// SIMATIC S7-200 project (STEP 7-Micro/WIN), CPU 224 REL 01.11

ORGANIZATION_BLOCK 主:OB1
TITLE=这个项目是基于CPU224的工业脉冲除尘控制系统。已经被实际应用于现实水泥厂布袋除尘器，提供给大家当福利了。
// 系统支持手动和自动两种喷吹模式，分别由I0.0和I0.1控制，手动和自动模式不能同时启用。
// 系统控制的物理设备包括手动喷吹启动按钮、自动喷吹启动按钮、喷吹模式选择开关、喷吹参数选择开关和多个脉冲阀。
// 操作员可以通过手动喷吹启动按钮触发一次手动喷吹，或者按下自动喷吹启动按钮进入自动喷吹模式。不过，手动喷吹启动按钮和自动喷吹启动按钮设计上需避免同时按下，以确保模式切换清晰且操作安全。当两个按钮都未按下时，所有脉冲阀保持关闭，系统停止喷吹，防止意外运行。
// 操作员还可以通过喷吹模式选择开关1、喷吹模式选择开关2和喷吹模式选择开关3的组合，将喷吹时间参数设置为2到9之间的特定值；通过喷吹参数选择开关1、喷吹参数选择开关2和喷吹参数选择开关3的组合，将喷吹间隔参数设置为61到201之间的特定值。喷吹时间参数和喷吹间隔参数分别控制每个脉冲阀的开启时间和阀门之间的等待时间。例如，在手动模式下，按下手动喷吹启动按钮后，系统从脉冲阀1到脉冲阀28依次喷吹，每个阀门按喷吹时间参数开启，间隔由喷吹间隔参数决定。系统通过喷吹状态保持继电器1至喷吹状态保持继电器53管理喷吹过程中的状态转换，确保顺序执行。
// 在自动模式下，系统启动后从脉冲阀1到脉冲阀28完成一次喷吹，周期结束后所有喷吹状态保持继电器和脉冲阀自动复位。而在任一模式下，喷吹完成后，所有喷吹状态保持继电器和脉冲阀都会复位，以保持系统状态的正确性。在手动模式下，喷吹周期完成后，所有喷吹状态保持继电器和脉冲阀复位，等待手动喷吹启动按钮的下一次触发。
// 
//  
BEGIN
Network 1 // 网络题目 (单行)
//  
// 网络注释
//  
// 
LD     SM0.1
R      M0.0, 60
R      T37, 26
R      T101, 30
R      Q0.0, 32
Network 2
LD     I0.0
AN     I0.1
CALL   SBR_0:SBR1
Network 3
LD     I0.1
AN     I0.0
CALL   SBR_1:SBR0
Network 4
LDN    I0.0
AN     I0.1
LPS
R      M0.0, 60
R      Q0.0, 32
R      T37, 26
R      T101, 30
AN     I0.2
AN     I0.3
A      I0.4
MOVW   +2, VW50
LRD
AN     I0.5
AN     I0.6
A      I0.7
MOVW   +61, VW52
LRD
AN     I0.2
A      I0.3
AN     I0.4
MOVW   +3, VW50
LRD
AN     I0.5
A      I0.6
AN     I0.7
MOVW   +81, VW52
LRD
AN     I0.2
A      I0.3
A      I0.4
MOVW   +4, VW50
LRD
AN     I0.5
A      I0.6
A      I0.7
MOVW   +101, VW52
LRD
A      I0.2
AN     I0.3
AN     I0.4
MOVW   +5, VW50
LRD
A      I0.5
AN     I0.6
AN     I0.7
MOVW   +121, VW52
LRD
A      I0.2
AN     I0.3
A      I0.4
MOVW   +6, VW50
LRD
A      I0.5
AN     I0.6
A      I0.7
MOVW   +141, VW52
LRD
A      I0.2
A      I0.3
AN     I0.4
MOVW   +7, VW50
LRD
A      I0.5
A      I0.6
AN     I0.7
MOVW   +161, VW52
LRD
A      I0.2
A      I0.3
A      I0.4
MOVW   +8, VW50
LPP
A      I0.5
A      I0.6
A      I0.7
MOVW   +181, VW52
Network 5
LDN    I0.0
AN     I0.1
LPS
AN     I0.2
AN     I0.3
AN     I0.4
MOVW   +9, VW50
LPP
AN     I0.5
AN     I0.6
AN     I0.7
MOVW   +201, VW52
END_ORGANIZATION_BLOCK

SUBROUTINE_BLOCK SBR_1:SBR0
TITLE= 
// 子程序注释
// 按 F1 获得帮助及举例程序
//  
BEGIN
Network 1 // 网络题目 (单行)
//  
// 网络注释
//  
// 
LD     I0.1
AN     M0.0
R      Q0.0, 28
S      Q0.0, 1
S      M0.0, 1
Network 2
LD     M0.0
A      Q0.0
TON    T37, VW50
Network 3
LDN    M0.1
A      T37
R      Q0.0, 1
R      T37, 1
S      M0.1, 1
Network 4
LD     M0.1
AN     Q0.0
TON    T101, VW52
Network 5
LD     T101
AN     M0.2
R      M0.1, 1
R      T101, 1
S      Q0.1, 1
S      M0.2, 1
Network 6
LD     M0.2
A      Q0.1
TON    T38, VW50
Network 7
LDN    M0.3
A      T38
R      Q0.1, 1
R      T38, 1
S      M0.3, 1
Network 8
LD     M0.3
AN     Q0.1
TON    T102, VW52
Network 9
LD     T102
AN     M0.4
R      M0.3, 1
R      T102, 1
S      Q0.2, 1
S      M0.4, 1
Network 10
LD     M0.4
A      Q0.2
TON    T39, VW50
Network 11
LDN    M0.5
A      T39
R      Q0.2, 1
R      T39, 1
S      M0.5, 1
Network 12
LD     M0.5
AN     Q0.2
TON    T103, VW52
Network 13
LD     T103
AN     M0.6
R      M0.5, 1
R      T103, 1
S      Q0.3, 1
S      M0.6, 1
Network 14
LD     M0.6
A      Q0.3
TON    T40, VW50
Network 15
LDN    M0.7
A      T40
R      Q0.3, 1
R      T40, 1
S      M0.7, 1
Network 16
LD     M0.7
AN     Q0.3
TON    T104, VW52
Network 17
LD     T104
AN     M1.0
R      M0.7, 1
R      T104, 1
S      Q0.4, 1
S      M1.0, 1
Network 18
LD     M1.0
A      Q0.4
TON    T41, VW50
Network 19
LDN    M1.1
A      T41
R      Q0.4, 1
R      T41, 1
S      M1.1, 1
Network 20
LD     M1.1
AN     Q0.4
TON    T105, VW52
Network 21
LD     T105
AN     M1.2
R      M1.1, 1
R      T105, 1
S      Q0.5, 1
S      M1.2, 1
Network 22
LD     M1.2
A      Q0.5
TON    T42, VW50
Network 23
LDN    M1.3
A      T42
R      Q0.5, 1
R      T42, 1
S      M1.3, 1
Network 24
LD     M1.3
AN     Q0.5
TON    T106, VW52
Network 25
LD     T106
AN     M1.6
R      M1.3, 1
R      T106, 1
S      Q0.6, 1
S      M1.6, 1
Network 26
LD     M1.6
A      Q0.6
TON    T43, VW50
Network 27
LDN    M1.7
A      T43
R      Q0.6, 1
R      T43, 1
S      M1.7, 1
Network 28
LD     M1.7
AN     Q0.6
TON    T107, VW52
Network 29
LD     T107
AN     M2.0
R      M1.7, 1
R      T107, 1
S      Q0.7, 1
S      M2.0, 1
Network 30
LD     M2.0
A      Q0.7
TON    T44, VW50
Network 31
LDN    M2.1
A      T44
R      Q0.7, 1
R      T44, 1
S      M2.1, 1
Network 32
LD     M2.1
AN     Q0.7
TON    T108, VW52
Network 33
LD     T108
AN     M2.2
R      M2.1, 1
R      T108, 1
S      Q1.0, 1
S      M2.2, 1
Network 34
LD     M2.2
A      Q1.0
TON    T45, VW50
Network 35
LDN    M2.3
A      T45
R      Q1.0, 1
R      T45, 1
S      M2.3, 1
Network 36
LD     M2.3
AN     Q1.0
TON    T109, VW52
Network 37
LD     T109
AN     M2.4
R      M2.3, 1
R      T109, 1
S      Q1.1, 1
S      M2.4, 1
Network 38
LD     M2.4
A      Q1.1
TON    T46, VW50
Network 39
LDN    M2.5
A      T46
R      Q1.1, 1
R      T46, 1
S      M2.5, 1
Network 40
LD     M2.5
AN     Q1.1
TON    T110, VW52
Network 41
LD     T110
AN     M2.6
R      M2.5, 1
R      T110, 1
S      Q2.0, 1
S      M2.6, 1
Network 42
LD     M2.6
A      Q2.0
TON    T47, VW50
Network 43
LDN    M2.7
A      T47
R      Q2.0, 1
R      T47, 1
S      M2.7, 1
Network 44
LD     M2.7
AN     Q2.0
TON    T111, VW52
Network 45
LD     T111
AN     M3.0
R      M2.7, 1
R      T111, 1
S      Q2.1, 1
S      M3.0, 1
Network 46
LD     M3.0
A      Q2.1
TON    T48, VW50
Network 47
LDN    M3.1
A      T48
R      Q2.1, 1
R      T48, 1
S      M3.1, 1
Network 48
LD     M3.1
AN     Q2.1
TON    T112, VW52
Network 49
LD     T112
AN     M3.2
R      M3.1, 1
R      T112, 1
S      Q2.2, 1
S      M3.2, 1
Network 50
LD     M3.2
A      Q2.2
TON    T49, VW50
Network 51
LDN    M3.3
A      T49
R      Q2.2, 1
R      T49, 1
S      M3.3, 1
Network 52
LD     M3.3
AN     Q2.2
TON    T113, VW52
Network 53
LD     T113
AN     M3.4
R      M3.3, 1
R      T113, 1
S      Q2.3, 1
S      M3.4, 1
Network 54
LD     M3.4
A      Q2.3
TON    T50, VW50
Network 55
LDN    M3.5
A      T50
R      Q2.3, 1
R      T50, 1
S      M3.5, 1
Network 56
LD     M3.5
AN     Q2.3
TON    T114, VW52
Network 57
LD     T114
AN     M3.6
R      M3.5, 1
R      T114, 1
S      Q2.4, 1
S      M3.6, 1
Network 58
LD     M3.6
A      Q2.4
TON    T51, VW50
Network 59
LDN    M3.7
A      T51
R      Q2.4, 1
R      T51, 1
S      M3.7, 1
Network 60
LD     M3.7
AN     Q2.4
TON    T115, VW52
Network 61
LD     T115
AN     M4.0
R      M3.7, 1
R      T115, 1
S      Q2.5, 1
S      M4.0, 1
Network 62
LD     M4.0
A      Q2.5
TON    T52, VW50
Network 63
LDN    M4.1
A      T52
R      Q2.5, 1
R      T52, 1
S      M4.1, 1
Network 64
LD     M4.1
AN     Q2.5
TON    T116, VW52
Network 65
LD     T116
AN     M4.2
R      M4.1, 1
R      T116, 1
S      Q2.6, 1
S      M4.2, 1
Network 66
LD     M4.2
A      Q2.6
TON    T53, VW50
Network 67
LDN    M4.3
A      T53
R      Q2.6, 1
R      T53, 1
S      M4.3, 1
Network 68
LD     M4.3
AN     Q2.6
TON    T117, VW52
Network 69
LD     T117
AN     M4.4
R      M4.3, 1
R      T117, 1
S      Q2.7, 1
S      M4.4, 1
Network 70
LD     M4.4
A      Q2.7
TON    T54, VW50
Network 71
LDN    M4.5
A      T54
R      Q2.7, 1
R      T54, 1
S      M4.5, 1
Network 72
LD     M4.5
AN     Q2.7
TON    T118, VW52
Network 73
LD     T118
AN     M4.6
R      M4.5, 1
R      T118, 1
S      Q3.0, 1
S      M4.6, 1
Network 74
LD     M4.6
A      Q3.0
TON    T55, VW50
Network 75
LDN    M4.7
A      T55
R      Q3.0, 1
R      T55, 1
S      M4.7, 1
Network 76
LD     M4.7
AN     Q3.0
TON    T119, VW52
Network 77
LD     T119
AN     M5.0
R      M4.7, 1
R      T119, 1
S      Q3.1, 1
S      M5.0, 1
Network 78
LD     M5.0
A      Q3.1
TON    T56, VW50
Network 79
LDN    M5.1
A      T56
R      Q3.1, 1
R      T56, 1
S      M5.1, 1
Network 80
LD     M5.1
AN     Q3.1
TON    T120, VW52
Network 81
LD     T120
AN     M5.2
R      M5.1, 1
R      T120, 1
S      Q3.2, 1
S      M5.2, 1
Network 82
LD     M5.2
A      Q3.2
TON    T57, VW50
Network 83
LDN    M5.3
A      T57
R      Q3.2, 1
R      T57, 1
S      M5.3, 1
Network 84
LD     M5.3
AN     Q3.2
TON    T121, VW52
Network 85
LD     T121
AN     M5.4
R      M5.3, 1
R      T121, 1
S      Q3.3, 1
S      M5.4, 1
Network 86
LD     M5.4
A      Q3.3
TON    T58, VW50
Network 87
LDN    M5.5
A      T58
R      Q3.3, 1
R      T58, 1
S      M5.5, 1
Network 88
LD     M5.5
AN     Q3.3
TON    T122, VW52
Network 89
LD     T122
AN     M5.6
R      M5.5, 1
R      T122, 1
S      M5.6, 1
S      Q3.4, 1
Network 90
LD     M5.6
A      Q3.4
TON    T59, VW50
Network 91
LDN    M5.7
A      T59
R      Q3.4, 1
R      T59, 1
S      M5.7, 1
Network 92
LD     M5.7
AN     Q3.4
TON    T123, VW52
Network 93
LD     T123
AN     M6.0
R      M5.7, 1
R      T123, 1
S      M6.0, 1
S      Q3.5, 1
Network 94
LD     M6.0
A      Q3.5
TON    T60, VW50
Network 95
LDN    M6.1
A      T60
R      Q3.5, 1
R      T60, 1
S      M6.1, 1
Network 96
LD     M6.1
AN     Q3.5
TON    T124, VW52
Network 97
LD     T124
AN     M6.2
R      M6.1, 1
R      T124, 1
S      M6.2, 1
S      Q3.6, 1
Network 98
LD     M6.2
A      Q3.6
TON    T61, VW50
Network 99
LDN    M6.3
A      T61
R      Q3.6, 1
R      T61, 1
S      M6.3, 1
Network 100
LD     M6.3
AN     Q3.6
TON    T125, VW52
Network 101
LD     T125
AN     M6.4
R      M6.3, 1
R      T125, 1
S      M6.4, 1
Network 102
LD     M6.4
R      M0.0, 53
R      Q0.0, 32
R      M6.4, 1
END_SUBROUTINE_BLOCK

SUBROUTINE_BLOCK SBR_0:SBR1
TITLE=
BEGIN
Network 1
LD     I0.0
AN     M0.0
R      Q0.0, 28
S      Q0.0, 1
S      M0.0, 1
Network 2
LD     M0.0
A      Q0.0
TON    T37, VW50
Network 3
LDN    M0.1
A      T37
R      Q0.0, 1
R      T37, 1
S      M0.1, 1
Network 4
LD     M0.1
AN     Q0.0
TON    T101, VW52
Network 5
LD     T101
AN     M0.2
R      M0.1, 1
R      T101, 1
S      Q0.1, 1
S      M0.2, 1
Network 6
LD     M0.2
A      Q0.1
TON    T38, VW50
Network 7
LDN    M0.3
A      T38
R      Q0.1, 1
R      T38, 1
S      M0.3, 1
Network 8
LD     M0.3
AN     Q0.1
TON    T102, VW52
Network 9
LD     T102
AN     M0.4
R      M0.3, 1
R      T102, 1
S      Q0.2, 1
S      M0.4, 1
Network 10
LD     M0.4
A      Q0.2
TON    T39, VW50
Network 11
LDN    M0.5
A      T39
R      Q0.2, 1
R      T39, 1
S      M0.5, 1
Network 12
LD     M0.5
AN     Q0.2
TON    T103, VW52
Network 13
LD     T103
AN     M0.6
R      M0.5, 1
R      T103, 1
S      Q0.3, 1
S      M0.6, 1
Network 14
LD     M0.6
A      Q0.3
TON    T40, VW50
Network 15
LDN    M0.7
A      T40
R      Q0.3, 1
R      T40, 1
S      M0.7, 1
Network 16
LD     M0.7
AN     Q0.3
TON    T104, VW52
Network 17
LD     T104
AN     M1.0
R      M0.7, 1
R      T104, 1
S      Q0.4, 1
S      M1.0, 1
Network 18
LD     M1.0
A      Q0.4
TON    T41, VW50
Network 19
LDN    M1.1
A      T41
R      Q0.4, 1
R      T41, 1
S      M1.1, 1
Network 20
LD     M1.1
AN     Q0.4
TON    T105, VW52
Network 21
LD     T105
AN     M1.2
R      M1.1, 1
R      T105, 1
S      Q0.5, 1
S      M1.2, 1
Network 22
LD     M1.2
A      Q0.5
TON    T42, VW50
Network 23
LDN    M1.3
A      T42
R      Q0.5, 1
R      T42, 1
S      M1.3, 1
Network 24
LD     M1.3
AN     Q0.5
TON    T106, VW52
Network 25
LD     T106
AN     M1.6
R      M1.3, 1
R      T106, 1
S      Q0.6, 1
S      M1.6, 1
Network 26
LD     M1.6
A      Q0.6
TON    T43, VW50
Network 27
LDN    M1.7
A      T43
R      Q0.6, 1
R      T43, 1
S      M1.7, 1
Network 28
LD     M1.7
AN     Q0.6
TON    T107, VW52
Network 29
LD     T107
AN     M2.0
R      M1.7, 1
R      T107, 1
S      Q0.7, 1
S      M2.0, 1
Network 30
LD     M2.0
A      Q0.7
TON    T44, VW50
Network 31
LDN    M2.1
A      T44
R      Q0.7, 1
R      T44, 1
S      M2.1, 1
Network 32
LD     M2.1
AN     Q0.7
TON    T108, VW52
Network 33
LD     T108
AN     M2.2
R      M2.1, 1
R      T108, 1
S      Q1.0, 1
S      M2.2, 1
Network 34
LD     M2.2
A      Q1.0
TON    T45, VW50
Network 35
LDN    M2.3
A      T45
R      Q1.0, 1
R      T45, 1
S      M2.3, 1
Network 36
LD     M2.3
AN     Q1.0
TON    T109, VW52
Network 37
LD     T109
AN     M2.4
R      M2.3, 1
R      T109, 1
S      Q1.1, 1
S      M2.4, 1
Network 38
LD     M2.4
A      Q1.1
TON    T46, VW50
Network 39
LDN    M2.5
A      T46
R      Q1.1, 1
R      T46, 1
S      M2.5, 1
Network 40
LD     M2.5
AN     Q1.1
TON    T110, VW52
Network 41
LD     T110
AN     M2.6
R      M2.5, 1
R      T110, 1
S      Q2.0, 1
S      M2.6, 1
Network 42
LD     M2.6
A      Q2.0
TON    T47, VW50
Network 43
LDN    M2.7
A      T47
R      Q2.0, 1
R      T47, 1
S      M2.7, 1
Network 44
LD     M2.7
AN     Q2.0
TON    T111, VW52
Network 45
LD     T111
AN     M3.0
R      M2.7, 1
R      T111, 1
S      Q2.1, 1
S      M3.0, 1
Network 46
LD     M3.0
A      Q2.1
TON    T48, VW50
Network 47
LDN    M3.1
A      T48
R      Q2.1, 1
R      T48, 1
S      M3.1, 1
Network 48
LD     M3.1
AN     Q2.1
TON    T112, VW52
Network 49
LD     T112
AN     M3.2
R      M3.1, 1
R      T112, 1
S      Q2.2, 1
S      M3.2, 1
Network 50
LD     M3.2
A      Q2.2
TON    T49, VW50
Network 51
LDN    M3.3
A      T49
R      Q2.2, 1
R      T49, 1
S      M3.3, 1
Network 52
LD     M3.3
AN     Q2.2
TON    T113, VW52
Network 53
LD     T113
AN     M3.4
R      M3.3, 1
R      T113, 1
S      Q2.3, 1
S      M3.4, 1
Network 54
LD     M3.4
A      Q2.3
TON    T50, VW50
Network 55
LDN    M3.5
A      T50
R      Q2.3, 1
R      T50, 1
S      M3.5, 1
Network 56
LD     M3.5
AN     Q2.3
TON    T114, VW52
Network 57
LD     T114
AN     M3.6
R      M3.5, 1
R      T114, 1
S      Q2.4, 1
S      M3.6, 1
Network 58
LD     M3.6
A      Q2.4
TON    T51, VW50
Network 59
LDN    M3.7
A      T51
R      Q2.4, 1
R      T51, 1
S      M3.7, 1
Network 60
LD     M3.7
AN     Q2.4
TON    T115, VW52
Network 61
LD     T115
AN     M4.0
R      M3.7, 1
R      T115, 1
S      Q2.5, 1
S      M4.0, 1
Network 62
LD     M4.0
A      Q2.5
TON    T52, VW50
Network 63
LDN    M4.1
A      T52
R      Q2.5, 1
R      T52, 1
S      M4.1, 1
Network 64
LD     M4.1
AN     Q2.5
TON    T116, VW52
Network 65
LD     T116
AN     M4.2
R      M4.1, 1
R      T116, 1
S      Q2.6, 1
S      M4.2, 1
Network 66
LD     M4.2
A      Q2.6
TON    T53, VW50
Network 67
LDN    M4.3
A      T53
R      Q2.6, 1
R      T53, 1
S      M4.3, 1
Network 68
LD     M4.3
AN     Q2.6
TON    T117, VW52
Network 69
LD     T117
AN     M4.4
R      M4.3, 1
R      T117, 1
S      Q2.7, 1
S      M4.4, 1
Network 70
LD     M4.4
A      Q2.7
TON    T54, VW50
Network 71
LDN    M4.5
A      T54
R      Q2.7, 1
R      T54, 1
S      M4.5, 1
Network 72
LD     M4.5
AN     Q2.7
TON    T118, VW52
Network 73
LD     T118
AN     M4.6
R      M4.5, 1
R      T118, 1
S      Q3.0, 1
S      M4.6, 1
Network 74
LD     M4.6
A      Q3.0
TON    T55, VW50
Network 75
LDN    M4.7
A      T55
R      Q3.0, 1
R      T55, 1
S      M4.7, 1
Network 76
LD     M4.7
AN     Q3.0
TON    T119, VW52
Network 77
LD     T119
AN     M5.0
R      M4.7, 1
R      T119, 1
S      Q3.1, 1
S      M5.0, 1
Network 78
LD     M5.0
A      Q3.1
TON    T56, VW50
Network 79
LDN    M5.1
A      T56
R      Q3.1, 1
R      T56, 1
S      M5.1, 1
Network 80
LD     M5.1
AN     Q3.1
TON    T120, VW52
Network 81
LD     T120
AN     M5.2
R      M5.1, 1
R      T120, 1
S      Q3.2, 1
S      M5.2, 1
Network 82
LD     M5.2
A      Q3.2
TON    T57, VW50
Network 83
LDN    M5.3
A      T57
R      Q3.2, 1
R      T57, 1
S      M5.3, 1
Network 84
LD     M5.3
AN     Q3.2
TON    T121, VW52
Network 85
LD     T121
AN     M5.4
R      M5.3, 1
R      T121, 1
S      Q3.3, 1
S      M5.4, 1
Network 86
LD     M5.4
A      Q3.3
TON    T58, VW50
Network 87
LDN    M5.5
A      T58
R      Q3.3, 1
R      T58, 1
S      M5.5, 1
Network 88
LD     M5.5
AN     Q3.3
TON    T122, VW52
Network 89
LD     T122
AN     M5.6
R      M5.5, 1
R      T122, 1
S      M5.6, 1
S      Q3.4, 1
Network 90
LD     M5.6
A      Q3.4
TON    T59, VW50
Network 91
LDN    M5.7
A      T59
R      Q3.4, 1
R      T59, 1
S      M5.7, 1
Network 92
LD     M5.7
AN     Q3.4
TON    T123, VW52
Network 93
LD     T123
AN     M6.0
R      M5.7, 1
R      T123, 1
S      M6.0, 1
S      Q3.5, 1
Network 94
LD     M6.0
A      Q3.5
TON    T60, VW50
Network 95
LDN    M6.1
A      T60
R      Q3.5, 1
R      T60, 1
S      M6.1, 1
Network 96
LD     M6.1
AN     Q3.5
TON    T124, VW52
Network 97
LD     T124
AN     M6.2
R      M6.1, 1
R      T124, 1
S      M6.2, 1
S      Q3.6, 1
Network 98
LD     M6.2
A      Q3.6
TON    T61, VW50
Network 99
LDN    M6.3
A      T61
R      Q3.6, 1
R      T61, 1
S      M6.3, 1
Network 100
LD     M6.3
AN     Q3.6
TON    T125, VW52
Network 101
LD     T125
AN     M6.4
R      M6.3, 1
R      T125, 1
S      M6.4, 1
Network 102
LD     M6.4
R      M0.0, 53
R      Q0.0, 32
R      M6.4, 1
END_SUBROUTINE_BLOCK
